// TIA Portal V19 export
ORGANIZATION_BLOCK "RACK_FLT"   // OB86, STL, RackOrStationFailure
TITLE = "Loss Of Rack Fault"
   VAR_TEMP
      OB86_EV_CLASS : Byte;   // 16#38/39 Event class 3
      OB86_FLT_ID : Byte;   // 16#C1/C4/C5, Fault identification code
      OB86_PRIORITY : Byte;   // Priority of OB Execution
      OB86_OB_NUMBR : Byte;   // 86 (Organization block 86, OB86)
      OB86_RESERVED_1 : Byte;   // Reserved for system
      OB86_RESERVED_2 : Byte;   // Reserved for system
      OB86_MDL_ADDR : Word;   // Base address of IM module in rack with fault
      OB86_RACKS_FLTD : Array[0..31] of Bool;   // Racks in fault
      OB86_DATE_TIME : Date_And_Time;   // Date and time OB86 started
   END_VAR
BEGIN

NETWORK
TITLE = Call system diagnostics block
      CALL  "RSE_FB", "RSE_DB";
END_ORGANIZATION_BLOCK
